TYPE ST_TouchProbe :
STRUCT
  // TouchProbe Function for EL Terminals
  ToPlc     : ST_TouchProbeSet;
  FromPlc   : ST_TouchProbeGet;
END_STRUCT
END_TYPE

(* stored: Version 1.1.0.1, ProductVersion 3.1.4024.12
   DUT ST_TouchProbe: Id {322daf40-c7cb-44d3-bee2-2d4a9fbb3256} *)
